FUNCTION_BLOCK FB_LogHandlerTests EXTENDS FB_TestSuite

//==============================================================
//MAIN TESTS
//==============================================================

testMain01_ReducedMaxImageSize_BufferOverflow();

//==============================================================
//NEGATIVE TESTS
//==============================================================

//==============================================================
//SEQUENCE TESTS
//==============================================================

//==============================================================
//OTHERS TESTS
//==============================================================

METHOD INTERNAL testMain01_ReducedMaxImageSize_BufferOverflow
VAR
	fbLogHandler			: FB_LOG_Handler;
	sLogMessage				: T_LongSTRING;
	
END_VAR
VAR_INST
	stEventDataUT				: ST_LOG_EventData;
END_VAR
TEST('testMain01_ReducedMaxImageSize_BufferOverflow');

stEventDataUT.bEnable := TRUE;
//stEventDataUT.sTimeStamp :=MID( F_SYSTEM_SystemTimeAsISO8601(gDevice.stMetsStatus.stCTDateTime.sSystemTime, gDevice.stMetsStatus.stCTDateTime.sUTCTimeZoneOffset ), 12, 12);
stEventDataUT.nMaxImageArraySize	:= 300;
sLogMessage := '$01ST=53;$02CT=10;DS=GZDNP5JOA3IL;OG=3;XP=-50;YP=50;AP=-88;CS=06.2;SC=0070;QS=3;PN=1;$03
					$01ST=53;$02CT=10;DS=N7E1Y89UNK3O;OG=3;XP=-50;YP=-50;AP=-88;CS=06.2;SC=0070;QS=3;PN=2;$03
					$01ST=53;$02CT=10;DS=JHWJXYFNX9DS;OG=3;XP=50;YP=50;AP=-88;CS=06.2;SC=0070;QS=3;PN=3;$03
					$01ST=53;$02CT=10;DS=XGBEZLBV8A9I;OG=3;XP=50;YP=-50;AP=-88;CS=06.2;SC=0070;QS=3;PN=4;$03';


fbLogHandler(
	_IsUsed:= TRUE, 
	bLogData:= TRUE , 
	sLogMessage:= sLogMessage , 
	stEventData:= stEventDataUT, 
	bDone=> , 
	bBufferOverflow=> );


AssertEquals_BOOL(Expected := TRUE, 
						Actual:= fbLogHandler.bBufferOverflow, 
						Message:= 'Buffer output state not as expected');
					
TEST_FINISHED();
END_METHOD

END_FUNCTION_BLOCK

(* stored: Version 1.1.0.1
   POU FB_LogHandlerTests: Id {f77039cd-321d-4c47-963c-91f86ae4e230}, SpecialFunc None
   Folder 01 Main: Id {28088f49-2207-4f0d-bd8e-933442717bd0}
   Folder 02 Negative: Id {71d7eb2b-832e-4d20-a52d-53857f5f4550}
   Method testMain01_ReducedMaxImageSize_BufferOverflow: Id {1393e1e3-b9c9-4caf-b40d-17cd59dab7b6} *)
